// TIA Portal V16 export
// export: Created 2024-12-03T15:41:43.988114Z, ExportSetting WithDefaults, DisplayName Totally Integrated Automation Portal, DisplayVersion V16 Update 6, DisplayName TIA Portal Version Control Interface, DisplayVersion V16 Update 2, DisplayName TIA Portal Openness, DisplayVersion V16 Update 6, DisplayName TIA Portal Teamcenter Gateway, DisplayVersion V16, DisplayName SINAMICS Startdrive Advanced, DisplayVersion V16 Update 5, DisplayName SINAMICS Startdrive G130, G150, S120, S150, SINAMICS MV, S210, DisplayVersion V16 Update 5, DisplayName SINAMICS Startdrive G110M, G120, G120C, G120D, G120P, G115D, DisplayVersion V16 Update 5, DisplayName STEP 7 Professional, DisplayVersion V16 Update 6, DisplayName STEP 7 Safety, DisplayVersion V16, DisplayName WinCC Advanced / Unified PC, DisplayVersion V16 Update 6
DATA_BLOCK "Tracking_DB"   // DB19
{ S7_Optimized_Access := 'FALSE' }
VERSION : 0.1
// stored: AutoNumber true, DBAccessibleFromOPCUA true, IsOnlyStoredInLoadMemory false, IsWriteProtectedInAS false
   VAR RETAIN
      TrackingId : UInt;
      EmptyTrackingSimple { S7_SetPoint := 'True'} : "Tracking_Simple_UDT_1";
      EmptyTracking { S7_SetPoint := 'True'} : "Tracking_UDT";
      TrackingLostIndex { S7_SetPoint := 'True'} : UInt := 59;
      BadReadIndex { S7_SetPoint := 'True'} : UInt := 57;
   END_VAR
BEGIN
END_DATA_BLOCK
